TYPE T_READING_LREAL :
STRUCT
	lrValue:	LREAL; 	// LREAL (DOUBLE)
END_STRUCT
END_TYPE

(* stored: Version 1.1.0.1, ProductVersion 3.1.4022.16
   DUT T_READING_LREAL: Id {d2583454-e599-412b-8b2f-3fdf3df926d6} *)
